// TIA Portal V20 export
VAR_GLOBAL   // PLC tag table "Constantes del QUIMAROX"
END_VAR
VAR_GLOBAL CONSTANT   // user constants
   CTE_MaxNumQuimarox : UInt := 5;
   CTE_MaxNumElementos : UInt := 50;
   CTE_InicioEventosQuimarox : UInt := 500;   // Num, Inicio de Eventos del Quimarox
   CTE_Evento_QCAR : UInt := 500;   // Evento Piene Cargado
   CTE_Evento_QDES : UInt := 501;   // Evento Peine DesCargado
   CTE_Evento_QPRE : UInt := 502;   // Evento Carga existente en el Peine
   CTE_Evento_QRST : UInt := 503;   // Evento Carga existente en el Peine en caso de Reset
   CTE_MaxNumVagones : UInt := 20;   // Peines
END_VAR
